FUNCTION_BLOCK CmdOneActuatorBasic (* Basic Function Block Type *)
  (* Standard: 61499-2 *)
  (* Version 0.0, 7/31/2024, Administrator, Schneider Electric, Template *)
  PACKAGE SE.Nereda;
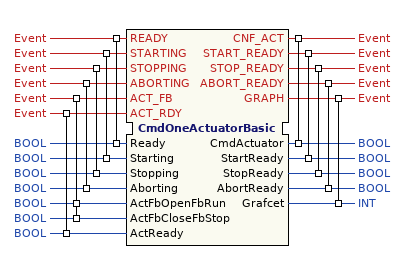
  EVENT_INPUT
    READY WITH Ready;
    STARTING WITH Starting; (* Normal Execution Request *)
    STOPPING WITH Stopping;
    ABORTING WITH Aborting;
    ACT_FB WITH ActFbOpenFbRun, ActFbCloseFbStop;
    ACT_RDY WITH ActReady;
  END_EVENT
  EVENT_OUTPUT
    CNF_ACT WITH CmdActuator; (* Execution Confirmation *)
    START_READY WITH StartReady;
    STOP_READY WITH StopReady;
    ABORT_READY WITH AbortReady;
    GRAPH WITH Grafcet;
  END_EVENT
  VAR_INPUT
    Ready : BOOL;
    Starting : BOOL; (* Input event qualifier *)
    Stopping : BOOL;
    Aborting : BOOL;
    ActFbOpenFbRun : BOOL;
    ActFbCloseFbStop : BOOL;
    ActReady : BOOL;
  END_VAR
  VAR_OUTPUT
    CmdActuator : BOOL; (* Output event qualifier *)
    StartReady : BOOL;
    StopReady : BOOL;
    AbortReady : BOOL;
    Grafcet : INT;
  END_VAR
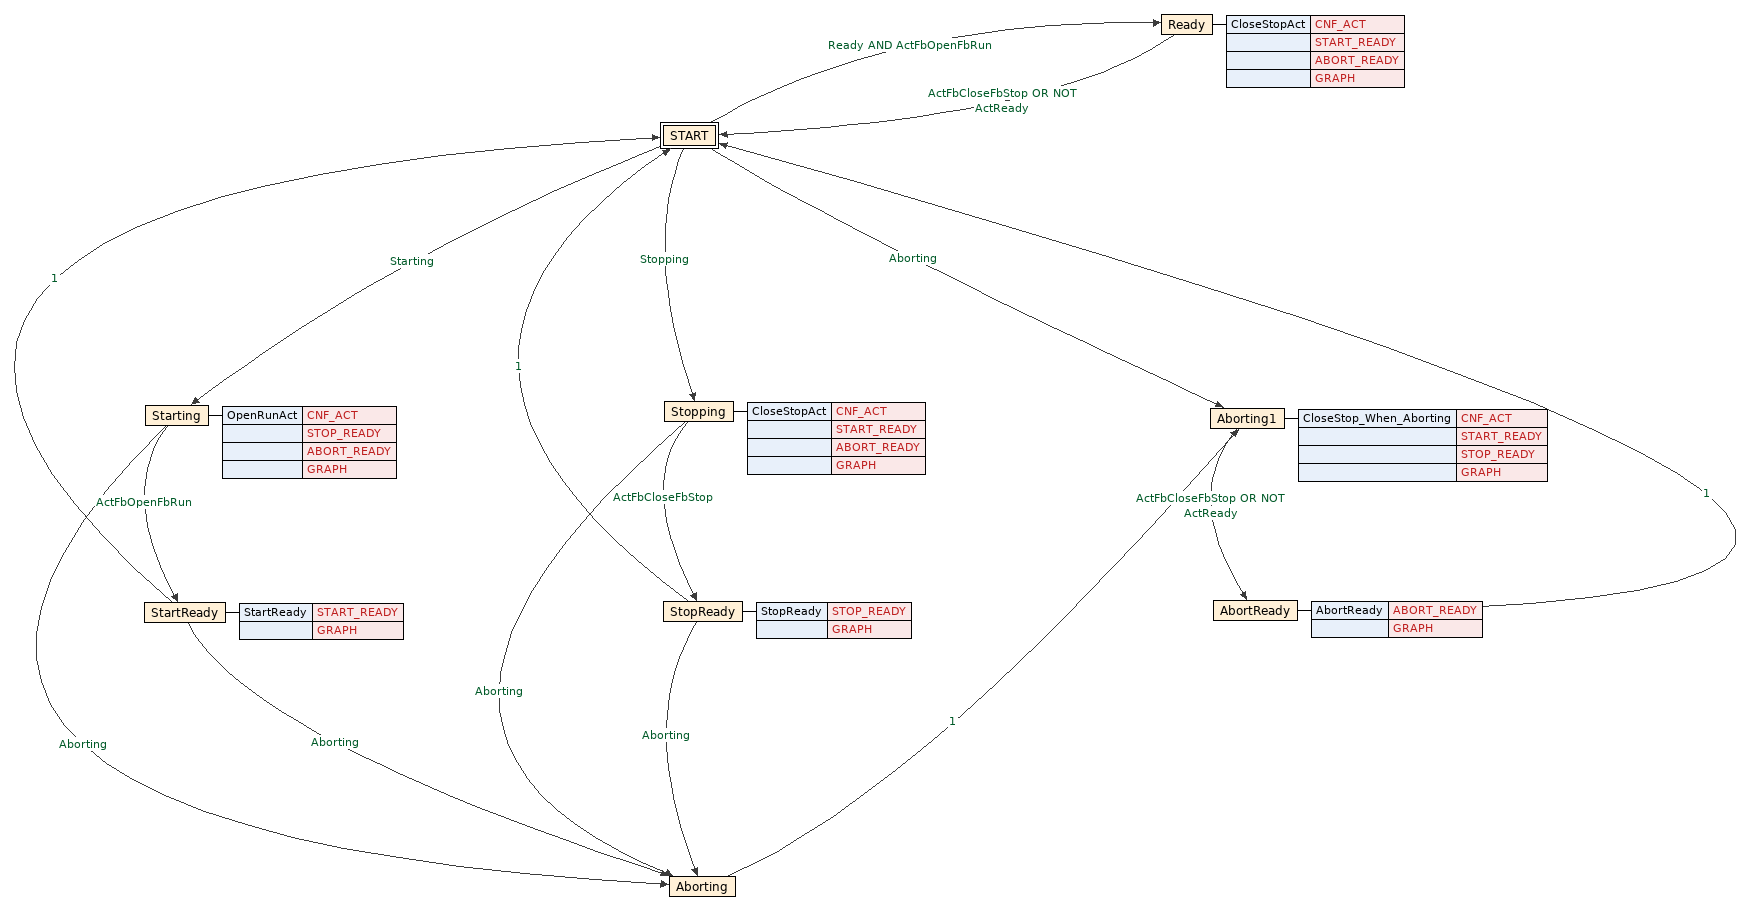
  EC_STATES
    START; (* Initial State *)
    Starting : OpenRunAct -> CNF_ACT, -> STOP_READY, -> ABORT_READY, -> GRAPH; (* Normal execution *)
    StartReady : StartReady -> START_READY, -> GRAPH;
    Stopping : CloseStopAct -> CNF_ACT, -> START_READY, -> ABORT_READY, -> GRAPH;
    StopReady : StopReady -> STOP_READY, -> GRAPH;
    Aborting1 : CloseStop_When_Aborting -> CNF_ACT, -> START_READY, -> STOP_READY, -> GRAPH;
    AbortReady : AbortReady -> ABORT_READY, -> GRAPH;
    Aborting;
    Ready : CloseStopAct -> CNF_ACT, -> START_READY, -> ABORT_READY, -> GRAPH;
  END_STATES
  EC_TRANSITIONS
    START TO Starting := Starting;
    Starting TO StartReady := ActFbOpenFbRun;
    StartReady TO START := 1;
    START TO Stopping := Stopping;
    Stopping TO StopReady := ActFbCloseFbStop;
    StopReady TO START := 1;
    Aborting1 TO AbortReady := ActFbCloseFbStop OR NOT ActReady;
    START TO Aborting1 := Aborting;
    AbortReady TO START := 1;
    Starting TO Aborting := Aborting;
    StartReady TO Aborting := Aborting;
    Aborting TO Aborting1 := 1;
    Stopping TO Aborting := Aborting;
    StopReady TO Aborting := Aborting;
    START TO Ready := Ready AND ActFbOpenFbRun;
    Ready TO START := ActFbCloseFbStop OR NOT ActReady;
  END_TRANSITIONS
  ALGORITHM OpenRunAct IN ST: (* Normally executed algorithm *)
;
Grafcet := 1;
CmdActuator := TRUE;
StopReady := FALSE;
AbortReady := FALSE;
  END_ALGORITHM
  ALGORITHM StartReady IN ST:
;
Grafcet := 2;
StartReady := TRUE;
  END_ALGORITHM
  ALGORITHM CloseStopAct IN ST:
;
Grafcet := 3;
CmdActuator := FALSE;
StartReady := FALSE;
AbortReady  := FALSE;
  END_ALGORITHM
  ALGORITHM StopReady IN ST:
;
Grafcet := 4;
StopReady := TRUE;
  END_ALGORITHM
  ALGORITHM CloseStop_When_Aborting IN ST:
;
Grafcet := 5;
CmdActuator := FALSE;
StartReady := FALSE;
StopReady := FALSE;
  END_ALGORITHM
  ALGORITHM AbortReady IN ST:
;
Grafcet := 6;
AbortReady := TRUE;
  END_ALGORITHM
END_FUNCTION_BLOCK
